// Block: PPrg_MAIN

DATA_BLOCK PPrg_MAIN
VERSION : 0.1
   NON_RETAIN
   VAR
      PIVOT : Array[1..PPRG_TOTAL_ARCHIVE_ITEMS] of Prg_Pivot;
      GET_ITF : Prg_GetITF;
      RWD : Struct
         EMPTY : PPrg_Data;
         UPDATE : PPrg_Data;
         GET : PPrg_Data;
         HMI : PPrg_Data;
         SCADA : PPrg_Data;
      END_STRUCT;
      HMI : Prg_HMI;
      SCADA : Prg_SCADA;
   END_VAR

BEGIN
   // No initialization required
END_DATA_BLOCK
